TYPE (* IEC61131-3, Table 14#5 *)
  (* Standard: 1131-3 *)
  (* Version 0.0, 1/8/2024, Cheyan, Schneider Electric, Template *)
  PACKAGE Main;
  {SET_ATTRIBUTE(nxtDataType, ZOG1cSCbfcbsYuYBrz+XyJSz6io8msJB/gnT/8b4foldDY4QobruYWY8+f3c9eli91haHrYjFi7Vq2buQ5wY+WxdAtWjZOjgL6UhThn+ty3WZ96iso1N/hkjBrZsGIjw)}
  SAV : STRUCT
    instMag : AnalogueValue;
    q : Quality;
  END_STRUCT;
END_TYPE
